(* PLC project TankLevelControl_TM241CE40T, PLCAutoPilot Tank Level Control - TM241CE40T 1.0 *)
(* stored: creationDateTime 2025-12-25T12:00:00, modificationDateTime 2025-12-25T12:00:00 *)

FUNCTION_BLOCK GVL_IO_TM241CE40T
  VAR
    DI_Tank1_LevelLow AT %IX0.0 : BOOL;  (* Tank 1 Low Level Switch (NC - TRUE when level OK) *)
    DI_Tank1_LevelHigh AT %IX0.1 : BOOL;  (* Tank 1 High Level Switch (NO - TRUE when high) *)
    DI_Tank2_LevelLow AT %IX0.2 : BOOL;  (* Tank 2 (RO) Low Level Switch *)
    DI_Tank2_LevelHigh AT %IX0.3 : BOOL;  (* Tank 2 (RO) High Level Switch *)
    DI_Start AT %IX0.4 : BOOL;  (* Start Push Button (NO) *)
    DI_Stop AT %IX0.5 : BOOL;  (* Stop Push Button (NC - TRUE when not pressed) *)
    DI_EStop AT %IX0.6 : BOOL;  (* Emergency Stop (NC - TRUE when not pressed) *)
    DI_Reset AT %IX0.7 : BOOL;  (* Fault Reset Push Button (NO) *)
    DI_Pump1_OL AT %IX0.8 : BOOL;  (* Pump 1 Overload (NC - TRUE when OK) *)
    DI_Pump2_OL AT %IX0.9 : BOOL;  (* Pump 2 Overload (NC - TRUE when OK) *)
    DI_Pump1_Run_FB AT %IX0.10 : BOOL;  (* Pump 1 Running Feedback (from contactor aux) *)
    DI_Pump2_Run_FB AT %IX0.11 : BOOL;  (* Pump 2 Running Feedback (from contactor aux) *)
    DI_Auto_Mode AT %IX0.12 : BOOL;  (* Auto/Manual Selector (TRUE = Auto) *)
    DI_Manual_Pump1 AT %IX0.13 : BOOL;  (* Manual Pump 1 Run (in Manual mode) *)
    DI_Manual_Pump2 AT %IX0.14 : BOOL;  (* Manual Pump 2 Run (in Manual mode) *)
    DI_Spare_15 AT %IX0.15 : BOOL;  (* Spare Input *)
    DI_Spare_16 AT %IX0.16 : BOOL;
    DI_Spare_17 AT %IX0.17 : BOOL;
    DI_Spare_18 AT %IX0.18 : BOOL;
    DI_Spare_19 AT %IX0.19 : BOOL;
    DI_Spare_20 AT %IX0.20 : BOOL;
    DI_Spare_21 AT %IX0.21 : BOOL;
    DI_Spare_22 AT %IX0.22 : BOOL;
    DI_Spare_23 AT %IX0.23 : BOOL;
    DO_Pump1 AT %QX0.0 : BOOL;  (* Pump 1 Contactor Output *)
    DO_Pump2 AT %QX0.1 : BOOL;  (* Pump 2 Contactor Output *)
    DO_Running_Light AT %QX0.2 : BOOL;  (* System Running Indicator (Green) *)
    DO_Fault_Light AT %QX0.3 : BOOL;  (* Fault Indicator (Red) *)
    DO_Tank1_Low_Alarm AT %QX0.4 : BOOL;  (* Tank 1 Low Level Alarm *)
    DO_Tank1_High_Alarm AT %QX0.5 : BOOL;  (* Tank 1 High Level Alarm *)
    DO_Tank2_Low_Alarm AT %QX0.6 : BOOL;  (* Tank 2 (RO) Low Level Alarm *)
    DO_Tank2_High_Alarm AT %QX0.7 : BOOL;  (* Tank 2 (RO) High Level Alarm *)
    DO_Pump1_Run_Light AT %QX0.8 : BOOL;  (* Pump 1 Running Indicator *)
    DO_Pump2_Run_Light AT %QX0.9 : BOOL;  (* Pump 2 Running Indicator *)
    DO_Auto_Mode_Light AT %QX0.10 : BOOL;  (* Auto Mode Indicator *)
    DO_Horn AT %QX0.11 : BOOL;  (* Alarm Horn Output *)
    DO_Spare_12 AT %QX0.12 : BOOL;  (* Spare Output *)
    DO_Spare_13 AT %QX0.13 : BOOL;
    DO_Spare_14 AT %QX0.14 : BOOL;
    DO_Spare_15 AT %QX0.15 : BOOL;
  END_VAR

            
(* I/O Mapping for TM241CE40T - 24 DI / 16 DO *)
            
          
END_FUNCTION_BLOCK

(* TANK LEVEL CONTROL PROGRAM FOR TM241CE40T ========================================== Controller: Schneider Electric Modicon M241 Model: TM241CE40T (24 DI / 16 DO) RUNGS: 0-2: Start/Stop/EStop Control 3: Auto/Manual Mode Selection 4-6: Pump 1 Control (Auto + Manual + Output) 7-9: Pump 2 Control (Auto + Manual + Output) 10-13: Status Indicators 14-17: Level Alarms (Low/High for both tanks) 18-22: Fault Detection and Reset *)
PROGRAM Tank_Control_TM241CE40T
  VAR
    System_Running : BOOL := FALSE;  (* System running flag *)
    Pump1_Cmd : BOOL := FALSE;
    Pump2_Cmd : BOOL := FALSE;
    Fault_Flag : BOOL := FALSE;
    Auto_Mode : BOOL := TRUE;
    Pump1_Timer : TON;
    Pump2_Timer : TON;
    Horn_Timer : TON;
  END_VAR
  VAR_INPUT
    Tank1_LevelLow AT %IX0.0 : BOOL;  (* Tank 1 Low Level (NC) *)
    Tank1_LevelHigh AT %IX0.1 : BOOL;  (* Tank 1 High Level (NO) *)
    Tank2_LevelLow AT %IX0.2 : BOOL;  (* Tank 2 Low Level (NC) *)
    Tank2_LevelHigh AT %IX0.3 : BOOL;  (* Tank 2 High Level (NO) *)
    PB_Start AT %IX0.4 : BOOL;
    PB_Stop AT %IX0.5 : BOOL;
    PB_EStop AT %IX0.6 : BOOL;
    PB_Reset AT %IX0.7 : BOOL;
    Pump1_OL AT %IX0.8 : BOOL;
    Pump2_OL AT %IX0.9 : BOOL;
    Pump1_FB AT %IX0.10 : BOOL;
    Pump2_FB AT %IX0.11 : BOOL;
    Sel_Auto AT %IX0.12 : BOOL;
    Man_Pump1 AT %IX0.13 : BOOL;
    Man_Pump2 AT %IX0.14 : BOOL;
  END_VAR
  VAR_OUTPUT
    Pump1_Out AT %QX0.0 : BOOL;
    Pump2_Out AT %QX0.1 : BOOL;
    Running_Light AT %QX0.2 : BOOL;
    Fault_Light AT %QX0.3 : BOOL;
    Tank1_Low_Alarm AT %QX0.4 : BOOL;
    Tank1_High_Alarm AT %QX0.5 : BOOL;
    Tank2_Low_Alarm AT %QX0.6 : BOOL;
    Tank2_High_Alarm AT %QX0.7 : BOOL;
    Pump1_Run_Light AT %QX0.8 : BOOL;
    Pump2_Run_Light AT %QX0.9 : BOOL;
    Auto_Light AT %QX0.10 : BOOL;
    Horn_Out AT %QX0.11 : BOOL;
  END_VAR

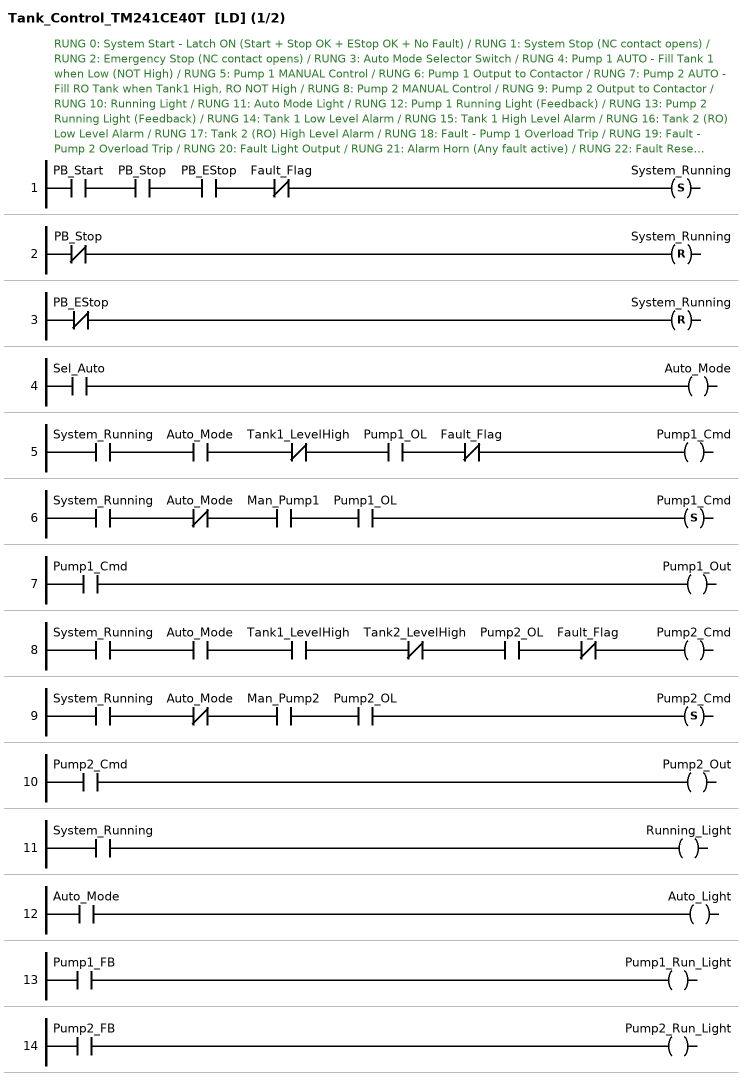
(* LD diagram, written out as Structured Text *)
(* RUNG 0: System Start - Latch ON (Start + Stop OK + EStop OK + No Fault) *)
IF PB_Start AND PB_Stop AND PB_EStop AND NOT Fault_Flag THEN System_Running := TRUE; END_IF;
(* RUNG 1: System Stop (NC contact opens) *)
IF NOT PB_Stop THEN System_Running := FALSE; END_IF;
(* RUNG 2: Emergency Stop (NC contact opens) *)
IF NOT PB_EStop THEN System_Running := FALSE; END_IF;
(* RUNG 3: Auto Mode Selector Switch *)
Auto_Mode := Sel_Auto;
(* RUNG 4: Pump 1 AUTO - Fill Tank 1 when Low (NOT High) *)
Pump1_Cmd := System_Running AND Auto_Mode AND NOT Tank1_LevelHigh AND Pump1_OL AND NOT Fault_Flag;
(* RUNG 5: Pump 1 MANUAL Control *)
IF System_Running AND NOT Auto_Mode AND Man_Pump1 AND Pump1_OL THEN Pump1_Cmd := TRUE; END_IF;
(* RUNG 6: Pump 1 Output to Contactor *)
Pump1_Out := Pump1_Cmd;
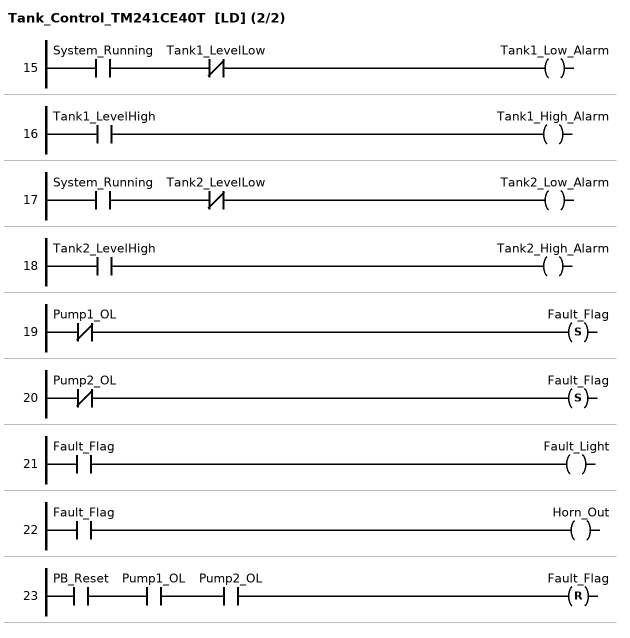
(* RUNG 7: Pump 2 AUTO - Fill RO Tank when Tank1 High, RO NOT High *)
Pump2_Cmd := System_Running AND Auto_Mode AND Tank1_LevelHigh AND NOT Tank2_LevelHigh AND Pump2_OL AND NOT Fault_Flag;
(* RUNG 8: Pump 2 MANUAL Control *)
IF System_Running AND NOT Auto_Mode AND Man_Pump2 AND Pump2_OL THEN Pump2_Cmd := TRUE; END_IF;
(* RUNG 9: Pump 2 Output to Contactor *)
Pump2_Out := Pump2_Cmd;
(* RUNG 10: Running Light *)
Running_Light := System_Running;
(* RUNG 11: Auto Mode Light *)
Auto_Light := Auto_Mode;
(* RUNG 12: Pump 1 Running Light (Feedback) *)
Pump1_Run_Light := Pump1_FB;
(* RUNG 13: Pump 2 Running Light (Feedback) *)
Pump2_Run_Light := Pump2_FB;
(* RUNG 14: Tank 1 Low Level Alarm *)
Tank1_Low_Alarm := System_Running AND NOT Tank1_LevelLow;
(* RUNG 15: Tank 1 High Level Alarm *)
Tank1_High_Alarm := Tank1_LevelHigh;
(* RUNG 16: Tank 2 (RO) Low Level Alarm *)
Tank2_Low_Alarm := System_Running AND NOT Tank2_LevelLow;
(* RUNG 17: Tank 2 (RO) High Level Alarm *)
Tank2_High_Alarm := Tank2_LevelHigh;
(* RUNG 18: Fault - Pump 1 Overload Trip *)
IF NOT Pump1_OL THEN Fault_Flag := TRUE; END_IF;
(* RUNG 19: Fault - Pump 2 Overload Trip *)
IF NOT Pump2_OL THEN Fault_Flag := TRUE; END_IF;
(* RUNG 20: Fault Light Output *)
Fault_Light := Fault_Flag;
(* RUNG 21: Alarm Horn (Any fault active) *)
Horn_Out := Fault_Flag;
(* RUNG 22: Fault Reset (Reset + OLs OK) *)
IF PB_Reset AND Pump1_OL AND Pump2_OL THEN Fault_Flag := FALSE; END_IF;
END_PROGRAM

CONFIGURATION TM241CE40T_Config
  RESOURCE TM241CE40T_Resource ON PLC
    TASK MAST(INTERVAL := T#10ms, PRIORITY := 1);
    PROGRAM Tank_Control_Instance WITH MAST : Tank_Control_TM241CE40T;
  END_RESOURCE
END_CONFIGURATION
